// TIA Portal V16 export
// export: Created 2025-10-06T17:54:38.1846884Z, ExportSetting WithDefaults, DisplayName Totally Integrated Automation Portal, DisplayVersion V16, DisplayName TIA Portal Version Control Interface, DisplayVersion V16, DisplayName TIA Portal Openness, DisplayVersion V16, DisplayName STEP 7 Professional, DisplayVersion V16, DisplayName STEP 7 Safety, DisplayVersion V16, DisplayName WinCC Advanced, DisplayVersion V16
DATA_BLOCK "OutputSinamics_DB"   // DB14
// stored: AutoNumber true, InstanceOfName OutputSinamics, OfSystemLibElement OutputSinamics, OfSystemLibVersion 2.3
"OutputSinamics"
   // VAR_INPUT
   //    TelNumber : Int;
   //    EnableDrive : Bool;
   //    StopMode : Int;
   //    OutErr : Bool;
   // END_VAR
   // VAR_OUTPUT
   //    OperationEnabled : Bool;
   //    Err_ID : Word;
   // END_VAR
   // VAR_IN_OUT
   //    Axis : Struct
   //       Sample_T : Real;
   //       AxisType : Bool;
   //       EncoderType : Bool;
   //       Sim : Bool;
   //       AxisLimitMax : Real;
   //       AxisLimitMin : Real;
   //       MaxVelocity : Real;
   //       MaxAcceleration : Real;
   //       MaxDeceleration : Real;
   //       MonTimeTargetAppr : Real;
   //       TargetRange : Real;
   //       StandstillRange : Real;
   //       MaxFollowingDist : Real;
   //       MonitorTargetAppr : Bool;
   //       SWLimitEnable : Bool;
   //       FactorP : Real;
   //       ManVelocity : Real;
   //       ManEnable : Bool;
   //       EmergencyDec : Real;
   //       InputModuleInAddr : Int;
   //       InputModuleOutAddr : Int;
   //       InputChannelNo : Int;
   //       StepsPerRev : DInt;
   //       DisplacementPerRev : Real;
   //       NumberRevs : Int;
   //       PolarityEncoder : Int;
   //       PositionOffset : DInt;
   //       OutputModuleOutAddr : Int;
   //       OutputModuleInAddr : Int;
   //       OutputChannelNo : Int;
   //       PolarityDrive : Int;
   //       DriveInputAtMaxVel : Real;
   //       OffsetCompensation : Real;
   //       DriveInputAt100 : Real;
   //       Override : Real;
   //       ActPosition : Real;
   //       FollowingDistance : Real;
   //       RemainingDistance : Real;
   //       NomVelocity : Real;
   //       ActVelocity : Real;
   //       Sync : Bool;
   //       Error : Bool;
   //       ErrorAck : Bool;
   //       AxisState : Int;
   //       Err : Struct
   //          SWLimitMinExceeded : Bool;
   //          SWLimitMaxExceeded : Bool;
   //          TargetErr : Bool;
   //          NoSync : Bool;
   //          DirectionErr : Bool;
   //          DataErr : Bool;
   //          StartErr : Bool;
   //          DistanceErr : Bool;
   //          MasterErr : Bool;
   //          bit09 : Bool;
   //          bit10 : Bool;
   //          bit11 : Bool;
   //          bit12 : Bool;
   //          bit13 : Bool;
   //          bit14 : Bool;
   //          bit15 : Bool;
   //          StoppedMotion : Bool;
   //          EnableDriveErr : Bool;
   //          FollowingDistErr : Bool;
   //          StandstillErr : Bool;
   //          TargetApproachErr : Bool;
   //          EncoderErr : Bool;
   //          OutputErr : Bool;
   //          ConfigErr : Bool;
   //          DriveErr : Bool;
   //          bit25 : Bool;
   //          bit26 : Bool;
   //          bit27 : Bool;
   //          bit28 : Bool;
   //          bit29 : Bool;
   //          bit30 : Bool;
   //          bit31 : Bool;
   //       END_STRUCT;
   //       Config : Struct
   //          Err_AxisLimit : Bool;
   //          Err_MaxVelocity : Bool;
   //          Err_MaxAcceleration : Bool;
   //          Err_MaxDeceleration : Bool;
   //          Err_MonTimeTargetAppr : Bool;
   //          Err_TargetRange : Bool;
   //          Err_StandstillRange : Bool;
   //          Err_MaxFollowingDist : Bool;
   //          Err_EmergencyDec : Bool;
   //          Err_StepsPerRev : Bool;
   //          Err_DisplacementPerRev : Bool;
   //          Err_NumberRevs : Bool;
   //          Err_PolarityEncoder : Bool;
   //          Err_PolarityDrive : Bool;
   //          Err_DriveInputAtMaxVel : Bool;
   //          Err_AxisLength : Bool;
   //          Err_EncoderRange : Bool;
   //          Err_MaxVelRotaryAxis : Bool;
   //          Err_DriveInputAt100 : Bool;
   //       END_STRUCT;
   //       EncoderValue : DInt;
   //       RefPoint : Real;
   //       OutVelocity : Real;
   //       LastNomPosition : Real;
   //       LastNomVelocity : Real;
   //       LastNomDeceleration : Real;
   //       InternalNomPosition : Real;
   //       InternalActPos : Real;
   //       InternalPosOffset : Real;
   //       aufl : Real;
   //       AchsLaenge : Real;
   //       AchsLaenge_DI : DInt;
   //       AbsGeberLaenge_DI : DInt;
   //       LageIstwert_DI : DInt;
   //       Coord : DInt;
   //       DoneRef : Bool;
   //       EinInitLaeuft : Bool;
   //       AusInitLaeuft : Bool;
   //       EinQuittungLaeuft : Bool;
   //       AusQuittungLaeuft : Bool;
   //       EintreiberFahrbereit : Bool;
   //       ExecRef : Int;
   //       VLastNomPosition : Real;
   //       VLastNomVelocity : Real;
   //       LastInternalPosOffset : Real;
   //       RundKorrektur : Real;
   //       LastRundKorrektur : Real;
   //       LengthUnit : String[4];
   //       InputModuleType : String[24];
   //       OutputModuleType : String[24];
   //       Init : Struct
   //          I0 : Bool;
   //          I1 : Bool;
   //          I2 : Bool;
   //          I3 : Bool;
   //          I4 : Bool;
   //          I5 : Bool;
   //          I6 : Bool;
   //          I7 : Bool;
   //          I8 : Bool;
   //          I9 : Bool;
   //          I10 : Bool;
   //          I11 : Bool;
   //          I12 : Bool;
   //          I13 : Bool;
   //          I14 : Bool;
   //          I15 : Bool;
   //          I16 : Bool;
   //          I17 : Bool;
   //          I18 : Bool;
   //          I19 : Bool;
   //          I20 : Bool;
   //          I21 : Bool;
   //          I22 : Bool;
   //          I23 : Bool;
   //          I24 : Bool;
   //          I25 : Bool;
   //          I26 : Bool;
   //          I27 : Bool;
   //          I28 : Bool;
   //          I29 : Bool;
   //          I30 : Bool;
   //          I31 : Bool;
   //       END_STRUCT;
   //    END_STRUCT;
   //    Init : Bool;
   // END_VAR
   // VAR RETAIN
   //    CONFIGURATION_DATA : Struct
   //       InputModuleInAddr : Int;
   //       OutputModuleOutAddr : Int;
   //       ProfiBus : Bool;
   //       ProfiNet : Bool;
   //       ID_Mastersystem : Int;
   //       Telegrammnumber : Int;
   //       TelegrFromInput : Int;
   //       InputFound : Bool;
   //       synchronous : Bool;
   //       invalid : Bool;
   //    END_STRUCT;
   //    Faktor : Real;
   //    OutputValue_R : Real;
   //    Lifecounter : Int;
   //    Addr_STW1 : Int;
   //    Addr_STW2 : Int;
   //    Addr_MRED : Int;
   //    Addr_ZSW1 : Int;
   //    Addr_ZSW2 : Int;
   //    Addr_MELDW : Int;
   //    Addr_NSOLL_B : Int;
   //    Addr_XERR : Int;
   //    Addr_KPC : Int;
   //    STW1_Offset : Int;
   //    STW2_Offset : Int;
   //    ZSW1_Offset : Int;
   //    ZSW2_Offset : Int;
   //    MRED_Offset : Int;
   //    MELDW_Offset : Int;
   //    NSOLL_B_Offset : Int;
   //    XERR_Offset : Int;
   //    KPC_Offset : Int;
   //    OutputValue : DInt;
   //    Quittungsautomat : Int;
   //    Einschaltautomat : Int;
   //    ZSW1 : Word;
   //    ZSW2 : Word;
   //    STW1 : Word;
   //    STW2 : Word;
   //    MELDW : Word;
   //    MRED : Word;
   //    wrong_OB : Bool;
   //    ERRORCODE : DWord;
   //    Virgin : Bool;
   //    FirstNormalRun : Bool;
   // END_VAR
BEGIN
END_DATA_BLOCK
